SUBAPPLICATION RobotStorageSensorInterlock (* Subapplication Type *)
  (* Standard: 61499-2 *)
  (* Version 1.0, 2021-08-10, dorofeev *)
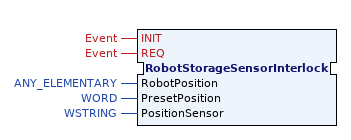
  EVENT_INPUT
    INIT;
    REQ;
  END_EVENT
  VAR_INPUT
    RobotPosition : ANY_ELEMENTARY;
    PresetPosition : WORD := 2;
    PositionSensor : WSTRING := 225.0.0.5:60000;
  END_VAR
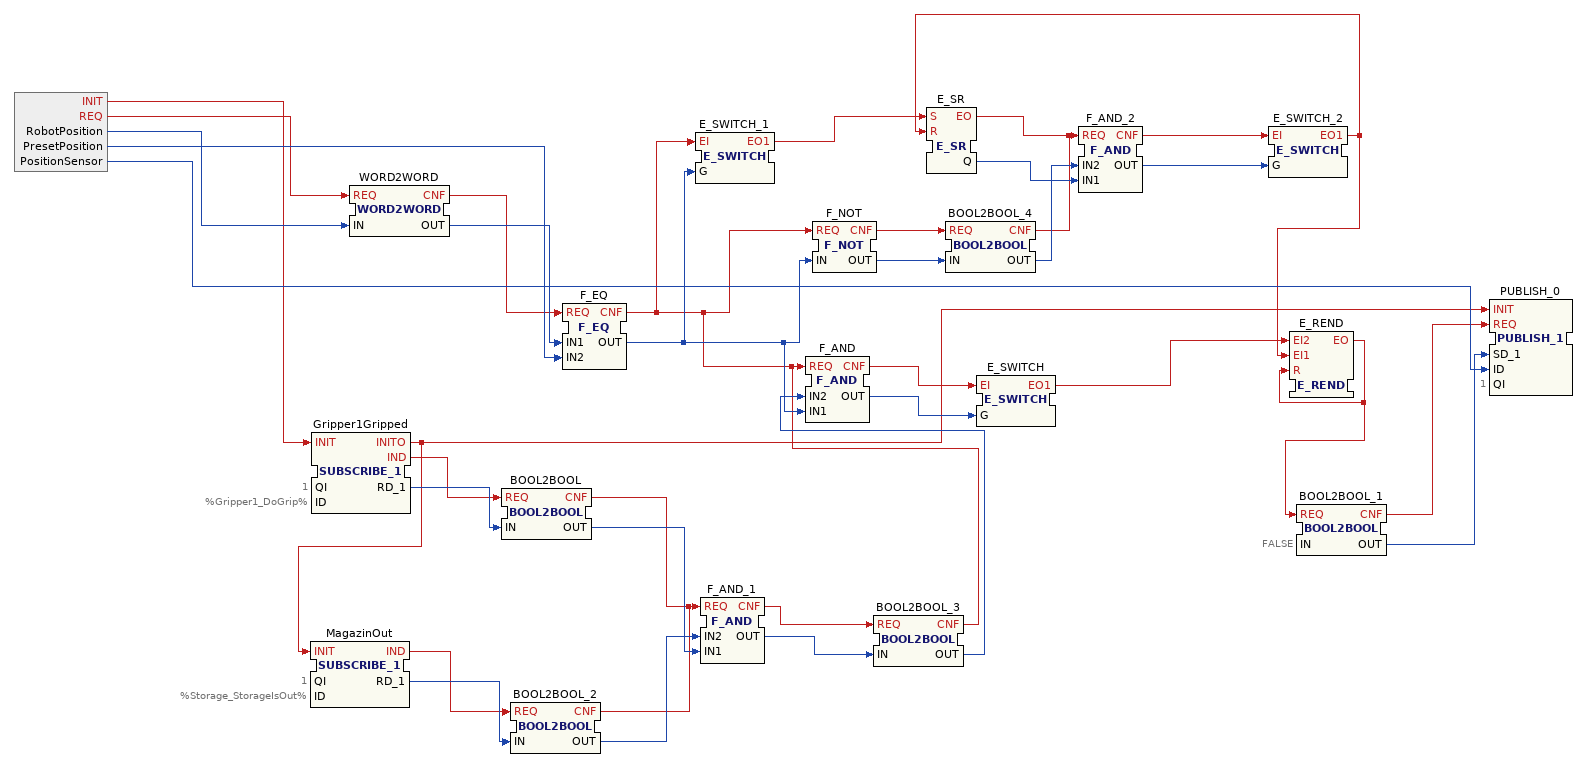
  FBS
    E_SWITCH : E_SWITCH;
    MagazinOut : SUBSCRIBE_1(QI := 1, ID := %Storage_StorageIsOut%);
    BOOL2BOOL : BOOL2BOOL;
    BOOL2BOOL_3 : BOOL2BOOL;
    Gripper1Gripped : SUBSCRIBE_1(QI := 1, ID := %Gripper1_DoGrip%);
    BOOL2BOOL_1 : BOOL2BOOL(IN := FALSE);
    F_EQ : F_EQ;
    BOOL2BOOL_2 : BOOL2BOOL;
    F_AND_1 : F_AND;
    F_AND : F_AND;
    E_REND : E_REND;
    PUBLISH_0 : PUBLISH_1(QI := 1);
    E_SR : E_SR;
    E_SWITCH_1 : E_SWITCH;
    F_AND_2 : F_AND;
    E_SWITCH_2 : E_SWITCH;
    F_NOT : F_NOT;
    BOOL2BOOL_4 : BOOL2BOOL;
    WORD2WORD : WORD2WORD;
  END_FBS
  EVENT_CONNECTIONS
    F_NOT.CNF TO BOOL2BOOL_4.REQ;
    F_EQ.CNF TO E_SWITCH_1.EI;
    Gripper1Gripped.INITO TO PUBLISH_0.INIT;
    MagazinOut.IND TO BOOL2BOOL_2.REQ;
    E_SR.EO TO F_AND_2.REQ;
    E_SWITCH_1.EO1 TO E_SR.S;
    F_AND.CNF TO E_SWITCH.EI;
    E_SWITCH.EO1 TO E_REND.EI2;
    BOOL2BOOL_4.CNF TO F_AND_2.REQ;
    BOOL2BOOL.CNF TO F_AND_1.REQ;
    Gripper1Gripped.INITO TO MagazinOut.INIT;
    Gripper1Gripped.IND TO BOOL2BOOL.REQ;
    F_EQ.CNF TO F_AND.REQ;
    BOOL2BOOL_1.CNF TO PUBLISH_0.REQ;
    E_REND.EO TO BOOL2BOOL_1.REQ;
    F_AND_2.CNF TO E_SWITCH_2.EI;
    E_SWITCH_2.EO1 TO E_REND.EI1;
    BOOL2BOOL_3.CNF TO F_AND.REQ;
    E_SWITCH_2.EO1 TO E_SR.R;
    F_AND_1.CNF TO BOOL2BOOL_3.REQ;
    E_REND.EO TO E_REND.R;
    BOOL2BOOL_2.CNF TO F_AND_1.REQ;
    F_EQ.CNF TO F_NOT.REQ;
    INIT TO Gripper1Gripped.INIT;
    REQ TO WORD2WORD.REQ;
    WORD2WORD.CNF TO F_EQ.REQ;
  END_CONNECTIONS
  DATA_CONNECTIONS
    F_EQ.OUT TO E_SWITCH_1.G;
    BOOL2BOOL_2.OUT TO F_AND_1.IN2;
    BOOL2BOOL_4.OUT TO F_AND_2.IN2;
    E_SR.Q TO F_AND_2.IN1;
    F_EQ.OUT TO F_NOT.IN;
    BOOL2BOOL_1.OUT TO PUBLISH_0.SD_1;
    F_AND.OUT TO E_SWITCH.G;
    BOOL2BOOL.OUT TO F_AND_1.IN1;
    F_NOT.OUT TO BOOL2BOOL_4.IN;
    Gripper1Gripped.RD_1 TO BOOL2BOOL.IN;
    BOOL2BOOL_3.OUT TO F_AND.IN2;
    F_EQ.OUT TO F_AND.IN1;
    F_AND_2.OUT TO E_SWITCH_2.G;
    MagazinOut.RD_1 TO BOOL2BOOL_2.IN;
    F_AND_1.OUT TO BOOL2BOOL_3.IN;
    PositionSensor TO PUBLISH_0.ID;
    WORD2WORD.OUT TO F_EQ.IN1;
    RobotPosition TO WORD2WORD.IN;
    PresetPosition TO F_EQ.IN2;
  END_CONNECTIONS
END_SUBAPPLICATION
